(* IEC 61131-3 sources: volt/packages/volt-lsp-iec/test-corpus/pro2193/Device/Plc Logic/Application/05 Global Var Lists, 12 files *)

(* ---- enumExchangeSets.dut ---- *)
{attribute 'qualified_only'}
{attribute 'strict'}
{attribute 'to_string'}
TYPE enumExchangeSets :
(
	Default
//	SingleCavSingleTakeover,
//	SingleCavDualTakeover,
//	FourCavDualTakeover,
//	TwoCavSingleTakeover
);
END_TYPE

// Please rename 'Default' to a more descriptive name.
// Check the type plate on the gripper how it is named.

// HINT!! Right-click on 'Default' -> Refactoring -> Rename ...

(* ---- RetainedVarsInBrinkRecipeType.dut ---- *)
// Retained variables that are saved in the Brink recipe. These are not changed when the customer picks a new recipe.
{attribute 'symbol' := 'readwrite'}
TYPE RetainedVarsInBrinkRecipeType :
STRUCT
	maximumAllowedCycleTime	: IntWithLimitsType	:=		// Time (sec) after which 'maximum allowed cycle time exceeded' alarm trips.
	(
		lowerLimit	:= 10,
		value		:= 30,
		upperLimit	:= 300,
		stepSize	:= 10
	);

	machineIdleShutoffTime	: IntWithLimitsType :=		// Time (min) when machine is inactive, shut off main air valve and vacuumpumps.
	(
		lowerLimit	:= 5,
		value		:= 30,
		upperLimit	:= 60 * 24 * 7,
		stepSize	:= 10
	);

	workingLightsTime		: IntWithLimitsType :=		// Time (min) that working lights will illuminate the inside of the machine.
	(
		lowerLimit	:= 5,
		value		:= 30,
		upperLimit	:= 60 * 24 * 7,
		stepSize	:= 5
	);

	// When the Xi Unit needs a label, and the magazine has no label ready: Wait for the label to be ready? Or check again the next cycle.
	// The process will wait for new labels for this time. After time-out the cycle continues without a label.
	cycleContinuesWithoutLabelsAfterTimeout		: RealWithLimitsType :=
	(
		lowerLimit	:= 0,						// Set to 0 to never wait for the magazine
		value		:= 10,
		upperLimit	:= 60.0 * 60.0 * 24,		// Set to 60*60*24 to wait the whole day
		stepSize	:= 1
	);

END_STRUCT
END_TYPE

(* ---- RetainedVarsInRecipeType.dut ---- *)
// Retained variables that are saved in the customer recipe
{attribute 'symbol' := 'readwrite'}
TYPE RetainedVarsInRecipeType :
STRUCT
	// Read only variables for safety. Vars can be changed by buttons in HMI program.
	{attribute 'symbol' := 'read'}	EnableIML					: BOOL;
	{attribute 'symbol' := 'read'}	EnableHMU					: BOOL;
	{attribute 'symbol' := 'read'}	EnableVision				: BOOL;
	{attribute 'symbol' := 'read'}	EnableSticker				: BOOL;

	ActiveExchangeSet			: enumExchangeSets;

	targetCycleTime				: REAL;	// The desired cycle time (sec) for this recipe. Used for statistics.

	productWeight				: REAL;	// Weight of a single product as measured by the customer (g).

	productPitch				: RealWithLimitsType :=		// Pitch between the products (mm).
	(
		lowerLimit	:= 0.1,
		value		:= 0.1,
		upperLimit	:= 100,
		stepSize	:= 0.1
	);

	productHeight				: RealWithLimitsType :=		// Height of a single product (mm).
	(
		lowerLimit	:= 1,
		value		:= 1,
		upperLimit	:= 500,
		stepSize	:= 2
	);

	{attribute 'symbol' := 'none'}	chainPos_XuUnit				: ARRAY[1..GVL_Constants.ChainProductsForXuUnit] OF UINT;
	{attribute 'symbol' := 'none'}	chainPos_Camera				: UINT;
	{attribute 'symbol' := 'none'}	chainPos_Reject				: ARRAY[1..GVL_Constants.ChainProductsForReject] OF UINT;
	{attribute 'symbol' := 'none'}	chainPos_ZUnit				: ARRAY[1..GVL_Constants.ChainProductsForZUnit] OF UINT;
	{attribute 'symbol' := 'none'}	chainPos_Sensor				: UINT;

END_STRUCT
END_TYPE

(* ---- GlobalVars.gvl ---- *)
{attribute 'symbol' := 'none'}
{attribute 'qualified_only'}
{attribute 'analysis' := '-33'}	// Unused Variable
VAR_GLOBAL
	Reset					: BOOL;					// Global reset active. From hardware button or input from visualisation
	EnableServoDrives		: BOOL;
	EnableMainvalve			: BOOL;
	manualControlRequested	: BOOL;					// Is high when a manual control button was pushed on the HMI

	BlinkerNormal			: BOOL;					// Global blinking bool. Default: high for 0,5 sec.
	BlinkerFast				: BOOL;					// Global fast blinker. Default: high for 0.2 sec.
	BlinkerPulseFast		: BOOL;					// Used by gates. Fast 0.1 sec. pulses
	BlinkerPulseSlow		: BOOL;					// Used by gates. Slow 0.1 sec. pulses

	EmergencyStopActive		: BOOL;					// Emergency-stop is active.

	debugTestBool1			: BOOL;
	debugTestBool2			: BOOL;
	debugTestInt1			: INT;
	debugTestInt2			: INT;
	debugTestInt3			: INT;
	debugTestInt4			: INT;
	debugTestInt5			: INT;
	debugSW					: ARRAY[0..9] OF StopwatchFB;

	// SUBRANGE not supported by VisiWinNet :(
	{attribute 'symbol' := 'readwrite'}	ActMouldLevels			: UINT(*(1..GVL_Constants.MaxMouldLevels)*)	:= GVL_Constants.MaxMouldLevels;
	{attribute 'symbol' := 'readwrite'}	ActProductsInX			: UINT(*(1..GVL_Constants.MaxProductsInX)*)	:= GVL_Constants.MaxProductsInX;
	{attribute 'symbol' := 'readwrite'}	ActProductsInY			: UINT(*(1..GVL_Constants.MaxProductsInY)*)	:= GVL_Constants.MaxProductsInY;
	ActProductsInMould		: UINT	:= ActMouldLevels * ActProductsInX * ActProductsInY;

	fbModuleManager			: ModuleManagerFB(name := 'SER');	// Keep a record of different kinds of modules in the machine.

	immediatelyGetNewLabels	: BOOL;					// In semi-auto mode, new labels are taken from magazine only AFTER the labels are inserted in the mould. This can overide that behaviouw.

	RuntimeConstants		: RuntimeConstantsType;	// For debugging: some constants about the PLC.

	// Options for debugging
	CheckBoundFunctionsThrowExceptions	: BOOL := FALSE;	// When the CheckBounds function has an error, the PLC is stopped. This makes troubleshooting easier.
	EnableDebugLogging					: BOOL := FALSE;	// Debug log messages are disabled and NOT logged to the PLC.
	EnableLoggingAllStateChanges		: BOOL := FALSE;	// Create a log message for every state change
	activeAlarmInstance					: STRING(80);		// For debugging: show id of module that has an alarm active
END_VAR

(* ---- GlobalVars_BFU.gvl ---- *)
{attribute 'symbol' := 'none'}
{attribute 'qualified_only'}
{attribute 'analysis' := '-33'}	// Unused Variable
VAR_GLOBAL
	Reset					: BOOL;					// Global reset active. From hardware button or input from visualisation
	EnableMainvalve			: BOOL;
	EnableServoDrives		: BOOL;

	fbModuleManager			: ModuleManagerFB(name := 'BFU');	// Keep a record of different kinds of modules in the machine.
END_VAR

(* ---- GVL_ComponentHardware.gvl ---- *)
(* This code is generated automatically *)
(* Don't change the content! *)

{attribute 'qualified_only'}
{attribute 'linkalways'}
VAR_GLOBAL
	//Controller
	Device 	: L_IC1P_ComponentHardware;

	//EtherCAT device
	L_i750_ZR 	: L_IC1P_ComponentHardware;
	L_i750_C2 	: L_IC1P_ComponentHardware;
	L_i750_M1 	: L_IC1P_ComponentHardware;
	L_i750_M2 	: L_IC1P_ComponentHardware;
	L_i750_Z 	: L_IC1P_ComponentHardware;
	L_i750_C1 	: L_IC1P_ComponentHardware;
	L_i750_Xi 	: L_IC1P_ComponentHardware;
	L_i750_Xu 	: L_IC1P_ComponentHardware;
	L_i950_Y 	: L_IC1P_ComponentHardware;
	RIO_M1 	: L_IC1P_ComponentHardware;
	RIO_Z1 	: L_IC1P_ComponentHardware;
	RIO_BFU 	: L_IC1P_ComponentHardware;
	FANUC_R_30iB_Plus 	: L_IC1P_ComponentHardware;

	//I/O module
	DI_30 	: L_IC1P_ComponentHardware;
	DI_31 	: L_IC1P_ComponentHardware;
	DI_32 	: L_IC1P_ComponentHardware;
	DI_33 	: L_IC1P_ComponentHardware;
	DQ_30 	: L_IC1P_ComponentHardware;
	DQ_31 	: L_IC1P_ComponentHardware;
	DQ_32 	: L_IC1P_ComponentHardware;
	DQ_33 	: L_IC1P_ComponentHardware;
	DQ_34 	: L_IC1P_ComponentHardware;
	DQ_35 	: L_IC1P_ComponentHardware;
	DQ_36 	: L_IC1P_ComponentHardware;
	DI_40 	: L_IC1P_ComponentHardware;
	DI_41 	: L_IC1P_ComponentHardware;
	DI_42 	: L_IC1P_ComponentHardware;
	DI_43 	: L_IC1P_ComponentHardware;
	DI_44 	: L_IC1P_ComponentHardware;
	DI_45 	: L_IC1P_ComponentHardware;
	DQ_40 	: L_IC1P_ComponentHardware;
	DQ_41 	: L_IC1P_ComponentHardware;
	DQ_42 	: L_IC1P_ComponentHardware;
	DQ_43 	: L_IC1P_ComponentHardware;
	DQ_44 	: L_IC1P_ComponentHardware;
	DQ_45 	: L_IC1P_ComponentHardware;
	DQ_46 	: L_IC1P_ComponentHardware;
	DI_50 	: L_IC1P_ComponentHardware;
	DI_51 	: L_IC1P_ComponentHardware;
	DI_52 	: L_IC1P_ComponentHardware;
	DI_53 	: L_IC1P_ComponentHardware;
	DI_54 	: L_IC1P_ComponentHardware;
	DQ_50 	: L_IC1P_ComponentHardware;
	DQ_51 	: L_IC1P_ComponentHardware;
	DQ_52 	: L_IC1P_ComponentHardware;
	DQ_53 	: L_IC1P_ComponentHardware;
	DQ_54 	: L_IC1P_ComponentHardware;

END_VAR

(* ---- GVL_Constants.gvl ---- *)
{attribute 'qualified_only'}
{attribute 'analysis' := '-33'}	// Unused Variable
VAR_GLOBAL CONSTANT
	MaxRejectReasonsMisc		: USINT			:= 1;		// IMM Euromap Reject, handle mounting reject, mould measurement reject, etc.
	MaxRejectReasonsCamera		: USINT			:= 7;		// Cam1 Reject, Cam2 Reject, etc.
	MaxRejectReasonsTotal		: USINT			:= MaxRejectReasonsMisc + MaxRejectReasonsCamera;

	MaxMouldLevels				: UINT			:= 1;		// In case of a stack mould, the number of mould faces (or levels)
	MaxProductsInX				: UINT			:= 3;		// Number of cavities in mould in X direction (horizontal)
	MaxProductsInY				: UINT			:= 4;		// Number of cavities in mould in Y direction (vertical)
	MaxProductsInMould			: UINT			:= MaxMouldLevels * MaxProductsInX * MaxProductsInY;	// Total number of cavities

	CavityStartIndex			: UINT			:= 1;											// Cavity numbering start index (usually 1)
	CavityEndIndex				: UINT			:= CavityStartIndex - 1 + MaxProductsInMould;	// Cavity numbering end index (usually the same as MaxProductsInMould)

	ChainProductsForXuUnit		: USINT			:= 4;
	ChainProductsForReject		: USINT			:= 1;
	ChainProductsForZUnit		: USINT			:= 6;
	ZUnitProductsForConveyor	: USINT			:= 12;

	ArmLength					: REAL			:= 895.0;	// Length of the arm/gripper in the drawer magazine in mm, normally 895 mm
	MaxAttemptsLabelTakeOut		: UINT			:= 1;		// Number of times the magazine attempts to take a label before assuming that the magazine is empty

	// Constants for Recipe Management
	RecipeDefinitionsCount		: INT			:= 3;		// Number of different recipe definitions
	AllRecipeDefinitions		: ARRAY[1..RecipeDefinitionsCount] OF STRING := ['Brink', 'Customer', 'Cassette'];	// Names of recipe definitions that are added to the Recipe Manager

	// Constants for Module Manager
	MaxNumberOfModules			: UINT			:= 40;		// Maximum amount of modules that the machine may have.
	MaxNumberOfStartableModules	: UINT			:= 20;		// Maximum amount of startable modules
	MaxNumberOfResettableModules: UINT			:= 20;		// Maximum amount of resettable modules
	MaxNumberOfServoDrives		: UINT			:= 20;		// Maximum amount of servo drives
	MaxNumberOfGates			: UINT			:= 10;		// Maximum amount of safety gates

	TimeLongest					: TIME			:= T#49D17H2M47S295MS;				// 4294967295
	DateTimeEarliest			: DATE_AND_TIME	:= DATE_AND_TIME#1970-1-1-00:00:00;	// 0
	DateTimeLatest				: DATE_AND_TIME	:= DATE_AND_TIME#2106-2-7-6:28:15;	// 4294967295

	RealSmallest				: REAL			:= -3.402823E+38;					// Smallest number
	RealLargest					: REAL			:=  3.402823E+38;					// Largest number
	LRealSmallest				: LREAL			:= -1.7976931348623157E+308;		// Smallest number
	LRealLargest				: LREAL			:=  1.7976931348623157E+308;		// Largest number
	DintSmallest				: DINT			:= -2147483648;						// Lower limit of DINT datatype
	DintLargest					: DINT			:=  2147483647;						// Upper limit of DINT datatype
	pi							: REAL			:= 3.14159274101257324;				// π
END_VAR

(* ---- GVL_Constants_BFU.gvl ---- *)
{attribute 'qualified_only'}
{attribute 'analysis' := '-33'}	// Unused Variable
VAR_GLOBAL CONSTANT
	MaxNumberOfStacksInBox		: UINT	:= 30;		// Maximum allowed number of stacks in the box

	// Constants for Module Manager
	MaxNumberOfModules			: UINT	:= 40;		// Maximum amount of modules that the machine may have.
	MaxNumberOfStartableModules	: UINT	:= 20;		// Maximum amount of startable modules
	MaxNumberOfResettableModules: UINT	:= 20;		// Maximum amount of resettable modules
	MaxNumberOfServoDrives		: UINT	:= 20;		// Maximum amount of servo drives
	MaxNumberOfGates			: UINT	:= 10;		// Maximum amount of safety gates
END_VAR

(* ---- GVL_Constants_Magazine.gvl ---- *)
{attribute 'qualified_only'}
VAR_GLOBAL CONSTANT
	MaxCassettes		: USINT := 16;
	MaxEnableValves		: USINT	:= 8;
	MaxAdjustValves		: USINT := 6;

	// Table defining all motors and directions for all possible combinations of label and cassette orientations
	OrientationTable	: ARRAY[1..64] OF OrientationEntry :=
	[
		(CassetteOrientation := enumOrientationType.Upright,	LabelOrientation := enumOrientationType.Upright,	Movement := enumMovementType.Up,	Motor := enumMotorsType.X,	Direction := enumdirection.Positive),
		(CassetteOrientation := enumOrientationType.Upright,	LabelOrientation := enumOrientationType.Upright,	Movement := enumMovementType.Down,	Motor := enumMotorsType.X,	Direction := enumDirection.Negative),
		(CassetteOrientation := enumOrientationType.Upright,	LabelOrientation := enumOrientationType.Upright,	Movement := enumMovementType.Left,	Motor := enumMotorsType.Y,	Direction := enumDirection.Negative),
		(CassetteOrientation := enumOrientationType.Upright,	LabelOrientation := enumOrientationType.Upright,	Movement := enumMovementType.Right,	Motor := enumMotorsType.Y,	Direction := enumDirection.Positive),
		(CassetteOrientation := enumOrientationType.Upright,	LabelOrientation := enumOrientationType.Right,		Movement := enumMovementType.Up,	Motor := enumMotorsType.Y,	Direction := enumDirection.Positive),
		(CassetteOrientation := enumOrientationType.Upright,	LabelOrientation := enumOrientationType.Right,		Movement := enumMovementType.Down,	Motor := enumMotorsType.Y,	Direction := enumDirection.Negative),
		(CassetteOrientation := enumOrientationType.Upright,	LabelOrientation := enumOrientationType.Right,		Movement := enumMovementType.Left,	Motor := enumMotorsType.X,	Direction := enumDirection.Positive),
		(CassetteOrientation := enumOrientationType.Upright,	LabelOrientation := enumOrientationType.Right,		Movement := enumMovementType.Right,	Motor := enumMotorsType.X,	Direction := enumDirection.Negative),
		(CassetteOrientation := enumOrientationType.Upright,	LabelOrientation := enumOrientationType.UpsideDown,	Movement := enumMovementType.Up,	Motor := enumMotorsType.X,	Direction := enumDirection.Negative),
		(CassetteOrientation := enumOrientationType.Upright,	LabelOrientation := enumOrientationType.UpsideDown,	Movement := enumMovementType.Down,	Motor := enumMotorsType.X,	Direction := enumDirection.Positive),
		(CassetteOrientation := enumOrientationType.Upright,	LabelOrientation := enumOrientationType.UpsideDown,	Movement := enumMovementType.Left,	Motor := enumMotorsType.Y,	Direction := enumDirection.Positive),
		(CassetteOrientation := enumOrientationType.Upright,	LabelOrientation := enumOrientationType.UpsideDown,	Movement := enumMovementType.Right,	Motor := enumMotorsType.Y,	Direction := enumDirection.Negative),
		(CassetteOrientation := enumOrientationType.Upright,	LabelOrientation := enumOrientationType.Left,		Movement := enumMovementType.Up,	Motor := enumMotorsType.Y,	Direction := enumDirection.Negative),
		(CassetteOrientation := enumOrientationType.Upright,	LabelOrientation := enumOrientationType.Left,		Movement := enumMovementType.Down,	Motor := enumMotorsType.Y,	Direction := enumDirection.Positive),
		(CassetteOrientation := enumOrientationType.Upright,	LabelOrientation := enumOrientationType.Left,		Movement := enumMovementType.Left,	Motor := enumMotorsType.X,	Direction := enumDirection.Negative),
		(CassetteOrientation := enumOrientationType.Upright,	LabelOrientation := enumOrientationType.Left,		Movement := enumMovementType.Right,	Motor := enumMotorsType.X,	Direction := enumDirection.Positive),
		(CassetteOrientation := enumOrientationType.Right,		LabelOrientation := enumOrientationType.Upright,	Movement := enumMovementType.Up,	Motor := enumMotorsType.Y,	Direction := enumDirection.Negative),
		(CassetteOrientation := enumOrientationType.Right,		LabelOrientation := enumOrientationType.Upright,	Movement := enumMovementType.Down,	Motor := enumMotorsType.Y,	Direction := enumDirection.Positive),
		(CassetteOrientation := enumOrientationType.Right,		LabelOrientation := enumOrientationType.Upright,	Movement := enumMovementType.Left,	Motor := enumMotorsType.X,	Direction := enumDirection.Negative),
		(CassetteOrientation := enumOrientationType.Right,		LabelOrientation := enumOrientationType.Upright,	Movement := enumMovementType.Right,	Motor := enumMotorsType.X,	Direction := enumDirection.Positive),
		(CassetteOrientation := enumOrientationType.Right,		LabelOrientation := enumOrientationType.Right,		Movement := enumMovementType.Up,	Motor := enumMotorsType.X,	Direction := enumDirection.Positive),
		(CassetteOrientation := enumOrientationType.Right,		LabelOrientation := enumOrientationType.Right,		Movement := enumMovementType.Down,	Motor := enumMotorsType.X,	Direction := enumDirection.Negative),
		(CassetteOrientation := enumOrientationType.Right,		LabelOrientation := enumOrientationType.Right,		Movement := enumMovementType.Left,	Motor := enumMotorsType.Y,	Direction := enumDirection.Negative),
		(CassetteOrientation := enumOrientationType.Right,		LabelOrientation := enumOrientationType.Right,		Movement := enumMovementType.Right,	Motor := enumMotorsType.Y,	Direction := enumDirection.Positive),
		(CassetteOrientation := enumOrientationType.Right,		LabelOrientation := enumOrientationType.UpsideDown,	Movement := enumMovementType.Up,	Motor := enumMotorsType.Y,	Direction := enumDirection.Positive),
		(CassetteOrientation := enumOrientationType.Right,		LabelOrientation := enumOrientationType.UpsideDown,	Movement := enumMovementType.Down,	Motor := enumMotorsType.Y,	Direction := enumDirection.Negative),
		(CassetteOrientation := enumOrientationType.Right,		LabelOrientation := enumOrientationType.UpsideDown,	Movement := enumMovementType.Left,	Motor := enumMotorsType.X,	Direction := enumDirection.Positive),
		(CassetteOrientation := enumOrientationType.Right,		LabelOrientation := enumOrientationType.UpsideDown,	Movement := enumMovementType.Right,	Motor := enumMotorsType.X,	Direction := enumDirection.Negative),
		(CassetteOrientation := enumOrientationType.Right,		LabelOrientation := enumOrientationType.Left,		Movement := enumMovementType.Up,	Motor := enumMotorsType.X,	Direction := enumDirection.Negative),
		(CassetteOrientation := enumOrientationType.Right,		LabelOrientation := enumOrientationType.Left,		Movement := enumMovementType.Down,	Motor := enumMotorsType.X,	Direction := enumDirection.Positive),
		(CassetteOrientation := enumOrientationType.Right,		LabelOrientation := enumOrientationType.Left,		Movement := enumMovementType.Left,	Motor := enumMotorsType.Y,	Direction := enumDirection.Positive),
		(CassetteOrientation := enumOrientationType.Right,		LabelOrientation := enumOrientationType.Left,		Movement := enumMovementType.Right,	Motor := enumMotorsType.Y,	Direction := enumDirection.Negative),
		(CassetteOrientation := enumOrientationType.UpsideDown,	LabelOrientation := enumOrientationType.Upright,	Movement := enumMovementType.Up,	Motor := enumMotorsType.X,	Direction := enumDirection.Negative),
		(CassetteOrientation := enumOrientationType.UpsideDown,	LabelOrientation := enumOrientationType.Upright,	Movement := enumMovementType.Down,	Motor := enumMotorsType.X,	Direction := enumDirection.Positive),
		(CassetteOrientation := enumOrientationType.UpsideDown,	LabelOrientation := enumOrientationType.Upright,	Movement := enumMovementType.Left,	Motor := enumMotorsType.Y,	Direction := enumDirection.Positive),
		(CassetteOrientation := enumOrientationType.UpsideDown,	LabelOrientation := enumOrientationType.Upright,	Movement := enumMovementType.Right,	Motor := enumMotorsType.Y,	Direction := enumDirection.Negative),
		(CassetteOrientation := enumOrientationType.UpsideDown,	LabelOrientation := enumOrientationType.Right,		Movement := enumMovementType.Up,	Motor := enumMotorsType.Y,	Direction := enumDirection.Negative),
		(CassetteOrientation := enumOrientationType.UpsideDown,	LabelOrientation := enumOrientationType.Right,		Movement := enumMovementType.Down,	Motor := enumMotorsType.Y,	Direction := enumDirection.Positive),
		(CassetteOrientation := enumOrientationType.UpsideDown,	LabelOrientation := enumOrientationType.Right,		Movement := enumMovementType.Left,	Motor := enumMotorsType.X,	Direction := enumDirection.Negative),
		(CassetteOrientation := enumOrientationType.UpsideDown,	LabelOrientation := enumOrientationType.Right,		Movement := enumMovementType.Right,	Motor := enumMotorsType.X,	Direction := enumDirection.Positive),
		(CassetteOrientation := enumOrientationType.UpsideDown,	LabelOrientation := enumOrientationType.UpsideDown,	Movement := enumMovementType.Up,	Motor := enumMotorsType.X,	Direction := enumDirection.Positive),
		(CassetteOrientation := enumOrientationType.UpsideDown,	LabelOrientation := enumOrientationType.UpsideDown,	Movement := enumMovementType.Down,	Motor := enumMotorsType.X,	Direction := enumDirection.Negative),
		(CassetteOrientation := enumOrientationType.UpsideDown,	LabelOrientation := enumOrientationType.UpsideDown,	Movement := enumMovementType.Left,	Motor := enumMotorsType.Y,	Direction := enumDirection.Negative),
		(CassetteOrientation := enumOrientationType.UpsideDown,	LabelOrientation := enumOrientationType.UpsideDown,	Movement := enumMovementType.Right,	Motor := enumMotorsType.Y,	Direction := enumDirection.Positive),
		(CassetteOrientation := enumOrientationType.UpsideDown,	LabelOrientation := enumOrientationType.Left,		Movement := enumMovementType.Up,	Motor := enumMotorsType.Y,	Direction := enumDirection.Positive),
		(CassetteOrientation := enumOrientationType.UpsideDown,	LabelOrientation := enumOrientationType.Left,		Movement := enumMovementType.Down,	Motor := enumMotorsType.Y,	Direction := enumDirection.Negative),
		(CassetteOrientation := enumOrientationType.UpsideDown,	LabelOrientation := enumOrientationType.Left,		Movement := enumMovementType.Left,	Motor := enumMotorsType.X,	Direction := enumDirection.Positive),
		(CassetteOrientation := enumOrientationType.UpsideDown,	LabelOrientation := enumOrientationType.Left,		Movement := enumMovementType.Right,	Motor := enumMotorsType.X,	Direction := enumDirection.Negative),
		(CassetteOrientation := enumOrientationType.Left,		LabelOrientation := enumOrientationType.Upright,	Movement := enumMovementType.Up,	Motor := enumMotorsType.Y,	Direction := enumDirection.Positive),
		(CassetteOrientation := enumOrientationType.Left,		LabelOrientation := enumOrientationType.Upright,	Movement := enumMovementType.Down,	Motor := enumMotorsType.Y,	Direction := enumDirection.Negative),
		(CassetteOrientation := enumOrientationType.Left,		LabelOrientation := enumOrientationType.Upright,	Movement := enumMovementType.Left,	Motor := enumMotorsType.X,	Direction := enumDirection.Positive),
		(CassetteOrientation := enumOrientationType.Left,		LabelOrientation := enumOrientationType.Upright,	Movement := enumMovementType.Right,	Motor := enumMotorsType.X,	Direction := enumDirection.Negative),
		(CassetteOrientation := enumOrientationType.Left,		LabelOrientation := enumOrientationType.Right,		Movement := enumMovementType.Up,	Motor := enumMotorsType.X,	Direction := enumDirection.Negative),
		(CassetteOrientation := enumOrientationType.Left,		LabelOrientation := enumOrientationType.Right,		Movement := enumMovementType.Down,	Motor := enumMotorsType.X,	Direction := enumDirection.Positive),
		(CassetteOrientation := enumOrientationType.Left,		LabelOrientation := enumOrientationType.Right,		Movement := enumMovementType.Left,	Motor := enumMotorsType.Y,	Direction := enumDirection.Positive),
		(CassetteOrientation := enumOrientationType.Left,		LabelOrientation := enumOrientationType.Right,		Movement := enumMovementType.Right,	Motor := enumMotorsType.Y,	Direction := enumDirection.Negative),
		(CassetteOrientation := enumOrientationType.Left,		LabelOrientation := enumOrientationType.UpsideDown,	Movement := enumMovementType.Up,	Motor := enumMotorsType.Y,	Direction := enumDirection.Negative),
		(CassetteOrientation := enumOrientationType.Left,		LabelOrientation := enumOrientationType.UpsideDown,	Movement := enumMovementType.Down,	Motor := enumMotorsType.Y,	Direction := enumDirection.Positive),
		(CassetteOrientation := enumOrientationType.Left,		LabelOrientation := enumOrientationType.UpsideDown,	Movement := enumMovementType.Left,	Motor := enumMotorsType.X,	Direction := enumDirection.Negative),
		(CassetteOrientation := enumOrientationType.Left,		LabelOrientation := enumOrientationType.UpsideDown,	Movement := enumMovementType.Right,	Motor := enumMotorsType.X,	Direction := enumDirection.Positive),
		(CassetteOrientation := enumOrientationType.Left,		LabelOrientation := enumOrientationType.Left,		Movement := enumMovementType.Up,	Motor := enumMotorsType.X,	Direction := enumDirection.Positive),
		(CassetteOrientation := enumOrientationType.Left,		LabelOrientation := enumOrientationType.Left,		Movement := enumMovementType.Down,	Motor := enumMotorsType.X,	Direction := enumDirection.Negative),
		(CassetteOrientation := enumOrientationType.Left,		LabelOrientation := enumOrientationType.Left,		Movement := enumMovementType.Left,	Motor := enumMotorsType.Y,	Direction := enumDirection.Negative),
		(CassetteOrientation := enumOrientationType.Left,		LabelOrientation := enumOrientationType.Left,		Movement := enumMovementType.Right,	Motor := enumMotorsType.Y,	Direction := enumDirection.Positive)
	];
END_VAR

(* ---- GVL_HC.gvl ---- *)
(* This code is generated automatically *)
(* Don't change the content! *)

{attribute 'qualified_only'}
{attribute 'linkalways'}
VAR_GLOBAL
	HcGroups : ARRAY [0..1] OF L_ETC_HC_GROUP;
END_VAR

(* ---- GVL_VacuumNumbers.gvl ---- *)
{attribute 'analysis' := '-33'}	// Unused Variable
VAR_GLOBAL CONSTANT
	// Use the constants below to access bits in any integer parameter
	AllVacuums			: WORD := 0;	// Ask all vacuums (parameter is zero)
	Vacuum00			: WORD := 0;	// Vacuum 0 (first bit) will not be in use! Vacuums start numbering from 1.
	Vacuum01			: WORD := 1;	// Ask vacuum 1 (or products belonging to vacuum 1)
	Vacuum02			: WORD := 2;	// Ask vacuum 2 (or products belonging to vacuum 2)
	Vacuum03			: WORD := 3;	// Ask vacuum 3 (or products belonging to vacuum 3)
	Vacuum04			: WORD := 4;	// Ask vacuum 4 (or products belonging to vacuum 4)
	Vacuum05			: WORD := 5;	// Ask vacuum 5 (or products belonging to vacuum 5)
	Vacuum06			: WORD := 6;	// Ask vacuum 6 (or products belonging to vacuum 6)
	Vacuum07			: WORD := 7;	// Ask vacuum 7 (or products belonging to vacuum 7)
	Vacuum08			: WORD := 8;	// Ask vacuum 8 (or products belonging to vacuum 8)
	Vacuum09			: WORD := 9;	// Ask vacuum 9 (or products belonging to vacuum 9)
	Vacuum10			: WORD := 10;	// Ask vacuum 10 (or products belonging to vacuum 10)
	Vacuum11			: WORD := 11;	// Ask vacuum 11 (or products belonging to vacuum 11)
	Vacuum12			: WORD := 12;	// Ask vacuum 12 (or products belonging to vacuum 12)
	Vacuum13			: WORD := 13;	// Ask vacuum 13 (or products belonging to vacuum 13)
	Vacuum14			: WORD := 14;	// Ask vacuum 14 (or products belonging to vacuum 14)
	Vacuum15			: WORD := 15;	// Ask vacuum 15 (or products belonging to vacuum 15)
END_VAR

// So to access the second bit in an integer, use like this:
// vacuumIndex.Vacuum01 := true;

// No 'qualified_only' attribute! Or bitaccess doesn't work.

(* ---- PersistentVars.gvl ---- *)
{attribute 'qualified_only'}
{attribute 'symbol' := 'readwrite'}
VAR_GLOBAL PERSISTENT RETAIN
	RecipeVars						: RetainedVarsInRecipeType;
	BrinkRecipeVars					: RetainedVarsInBrinkRecipeType;

	disableBuzzer					: BOOL;					// Permanently disable the buzzer output

	// SUBRANGE not supported by VisiWinNet :(
	usiGlobalSERSpeed				: USINT(*(1..100)*) := 50;	// Limit speed of all drives in the SER robot (0 to 100%)
	usiGlobalBFUSpeed				: USINT(*(1..100)*) := 50;	// Limit speed of all drives in the BFU robot (0 to 100%)

	DisableVacuumWithAirButton		: BOOL := FALSE;
	DisableVacuumPump2				: BOOL;

	{attribute 'symbol' := 'none'}	vacuumPumpRunningTime		: UDINT;				// Total time the vacuumpump has been running.
	{attribute 'symbol' := 'none'}	vacuumPumpNumberOfStarts	: UDINT;				// Total number of times the vacuumpump has been started.
	{attribute 'symbol' := 'none'}	Statistics					: ARRAY[1..ProductionStatsFB.NumberOfStatisticSets] OF ProductionStatsType;

	rejectReasonDescriptions		: ARRAY[1..GVL_Constants.MaxRejectReasonsTotal] OF STRING(40) :=
	[
		'IMM Euromap Reject',		// 1
		'Cam 1 Reject',				// 2
		'Cam 2 Reject',				// 3
		'Cam 3 Reject',				// 4
		'Cam 4 Reject',				// 5
		'Cam 5 Reject',				// 6
		'Cam 6 Reject',				// 7
		'Cam 7 Reject'				// 8
	];

	{attribute 'symbol' := 'none'}	cavityAliases				: ARRAY[GVL_Constants.CavityStartIndex..GVL_Constants.CavityEndIndex] OF STRING(20);

	// Generated instance path of persistent variable
	CassetteAdjustments.Data: ARRAY [1..CassetteAdjustments.usiNumberOfUnits] OF ARRAY [enumDrawer.Upper..enumDrawer.Lower, 1..GVL_Constants_Magazine.MaxCassettes] OF CassettePosition;
	// Generated instance path of persistent variable
	CassetteAdjustments.SwitchCountEnable: ARRAY [1..CassetteAdjustments.usiNumberOfUnits] OF ARRAY [enumDrawer.Upper..enumDrawer.Lower, 1..GVL_Constants_Magazine.MaxEnableValves] OF UDINT;
	// Generated instance path of persistent variable
	CassetteAdjustments.SwitchCountAdjust: ARRAY [1..CassetteAdjustments.usiNumberOfUnits] OF ARRAY [enumDrawer.Upper..enumDrawer.Lower, 1..GVL_Constants_Magazine.MaxAdjustValves] OF UDINT;
	// Generated instance path of persistent variable
	CassetteAdjustments.SwitchCountCassette: ARRAY [1..CassetteAdjustments.usiNumberOfUnits] OF ARRAY [enumDrawer.Upper..enumDrawer.Lower, 1..GVL_Constants_Magazine.MaxCassettes] OF ARRAY [enumMotorsType.X1..enumMotorsType.Y] OF UDINT;
	// Generated instance path of persistent variable
	CassetteAdjustments.ActualCassettePosition: ARRAY [1..CassetteAdjustments.usiNumberOfUnits] OF ARRAY [enumDrawer.Upper..enumDrawer.Lower, 1..GVL_Constants_Magazine.MaxCassettes] OF CassettePosition;
	// Generated instance path of persistent variable
	CassetteAdjustments.TargetCassettePosition: ARRAY [1..CassetteAdjustments.usiNumberOfUnits] OF ARRAY [enumDrawer.Upper..enumDrawer.Lower, 1..GVL_Constants_Magazine.MaxCassettes] OF CassettePosition;
	// Generated instance path of persistent variable
	RecipeControl.activeRecipe: ARRAY [1..GVL_Constants.RecipeDefinitionsCount] OF STRING(80);
	// Generated instance path of persistent variable
	RecipeControl.MetaData: ARRAY [1..GVL_Constants.RecipeDefinitionsCount] OF RecipeMetaDataType;
	// Generated instance path of persistent variable
	Fanucs.Data: ARRAY [1..Fanucs.usiNumberOfUnits] OF FanucUnitBase_Data;
	// Generated instance path of persistent variable
	Fanucs.DataProject: ARRAY [1..Fanucs.usiNumberOfUnits] OF FanucUnit_Data;
	// Generated instance path of persistent variable
	Fanucs.GripperStatus: ARRAY [1..Fanucs.usiNumberOfUnits] OF StackStatusType;
	// Generated instance path of persistent variable
	YUnits.Data: ARRAY [1..YUnits.usiNumberOfUnits] OF YUnit_Default_Data;
	// Generated instance path of persistent variable
	YUnits.DataBrink: ARRAY [1..YUnits.usiNumberOfUnits] OF DataBrinkType;
	// Generated instance path of persistent variable
	YUnits.coveredDistance: ARRAY [1..YUnits.usiNumberOfUnits] OF UDINT;
	// Generated instance path of persistent variable
	XuUnits.Data: ARRAY [1..XuUnits.usiNumberOfUnits] OF XuUnit_Default_Data;
	// Generated instance path of persistent variable
	XuUnits.DataProject: ARRAY [1..XuUnits.usiNumberOfUnits] OF XuUnit_ForChain_Data;
	// Generated instance path of persistent variable
	XuUnits.DataBrink: ARRAY [1..XuUnits.usiNumberOfUnits] OF DataBrinkType;
	// Generated instance path of persistent variable
	XuUnits.coveredDistance: ARRAY [1..XuUnits.usiNumberOfUnits] OF UDINT;
	// Generated instance path of persistent variable
	ZUnits.Data: ARRAY [1..ZUnits.usiNumberOfUnits] OF ZUnit_Base_Data;
	// Generated instance path of persistent variable
	ZUnits.DataProject: ARRAY [1..ZUnits.usiNumberOfUnits] OF ZUnit_ForChainWithServoRotate_Data;
	// Generated instance path of persistent variable
	ZUnits.DataBrink: ARRAY [1..ZUnits.usiNumberOfUnits] OF DataBrinkType;
	// Generated instance path of persistent variable
	ZUnits.coveredDistance: ARRAY [1..ZUnits.usiNumberOfUnits] OF UDINT;
	// Generated instance path of persistent variable
	XiUnits.Data: ARRAY [1..XiUnits.usiNumberOfUnits] OF XiUnit_Default_Data;
	// Generated instance path of persistent variable
	XiUnits.DataProject: ARRAY [1..XiUnits.usiNumberOfUnits] OF XiUnit_Data;
	// Generated instance path of persistent variable
	XiUnits.DataBrink: ARRAY [1..XiUnits.usiNumberOfUnits] OF DataBrinkType;
	// Generated instance path of persistent variable
	XiUnits.coveredDistance: ARRAY [1..XiUnits.usiNumberOfUnits] OF UDINT;
	// Generated instance path of persistent variable
	ZRUnits.Data: ARRAY [1..ZRUnits.usiNumberOfUnits] OF ZRUnit_Default_Data;
	// Generated instance path of persistent variable
	ZRUnits.DataBrink: ARRAY [1..ZRUnits.usiNumberOfUnits] OF DataBrinkType;
	// Generated instance path of persistent variable
	ZRUnits.coveredDistance: ARRAY [1..ZRUnits.usiNumberOfUnits] OF UDINT;
	// Generated instance path of persistent variable
	Conveyors.Data: ARRAY [1..Conveyors.usiNumberOfUnits] OF Conveyor_Servo_Data;
	// Generated instance path of persistent variable
	Conveyors.DataBrink: ARRAY [1..Conveyors.usiNumberOfUnits] OF DataBrinkType;
	// Generated instance path of persistent variable
	Conveyors.DataReject: ARRAY [1..Conveyors.usiNumberOfUnits] OF Conveyor_Reject_Data;
	// Generated instance path of persistent variable
	Conveyors.coveredDistance: ARRAY [1..Conveyors.usiNumberOfUnits] OF UDINT;
	// Generated instance path of persistent variable
	Chains.Data: ARRAY [1..Chains.usiNumberOfUnits] OF ChainBase_Data;
	// Generated instance path of persistent variable
	Chains.DataProject: ARRAY [1..Chains.usiNumberOfUnits] OF Chain_WithCarrierPlates_Data;
	// Generated instance path of persistent variable
	Chains.DataBrink: ARRAY [1..Chains.usiNumberOfUnits] OF DataBrinkType;
	// Generated instance path of persistent variable
	Chains.coveredDistance: ARRAY [1..Chains.usiNumberOfUnits] OF UDINT;
	// Generated instance path of persistent variable
	Magazines.Data: ARRAY [1..Magazines.usiNumberOfUnits] OF Magazine_Data;
	// Generated instance path of persistent variable
	Magazines.DataMotors: ARRAY [1..Magazines.usiNumberOfUnits] OF MagazineMotors_Drawer_Data;
	// Generated instance path of persistent variable
	Magazines.DataBrink: ARRAY [1..Magazines.usiNumberOfUnits] OF MagazineMotors_Drawer_BrinkData;
	// Generated instance path of persistent variable
	Magazines.coveredDistance: ARRAY [1..Magazines.usiNumberOfUnits] OF ARRAY [PickPlaceAxesNames.A1..PickPlaceAxesNames.A2] OF UDINT;
	// Generated instance path of persistent variable
	InjectionMouldingMachine.Data: IMM_Data;
	// Generated instance path of persistent variable
	ProcessModules.XYControlData: ARRAY [1..ProcessModules.numberOfXYControls] OF XYControl_Data;
	// Generated instance path of persistent variable
	LabelSuppliers.Data: ARRAY [1..LabelSuppliers.usiNumberOfUnits] OF DrawerMagazine_Data;
	// Generated instance path of persistent variable
	VisionSystems.Data: ARRAY [1..VisionSystems.usiNumberOfUnits] OF VisionSystem_Base_Data;
	// Generated instance path of persistent variable
	VisionSystems.DataProject: ARRAY [1..VisionSystems.usiNumberOfUnits] OF VisionSystem_Mevisco_Data;
	// Generated instance path of persistent variable
	RejectStations.Data: ARRAY [1..RejectStations.usiNumberOfUnits] OF RejectStation_Base_Data;
	// Generated instance path of persistent variable
	RejectStations.DataProject: ARRAY [1..RejectStations.usiNumberOfUnits] OF RejectStation_WithBlowOff_Data;
	// Generated instance path of persistent variable
	BufferRacks.Data: ARRAY [1..BufferRacks.usiNumberOfUnits] OF BufferRack_Data;
	// Generated instance path of persistent variable
	BufferRacks.BufferStackStatus: ARRAY [1..BufferRacks.usiNumberOfUnits] OF StackStatusType;
	// Generated instance path of persistent variable
	BufferRacks.BufferStackIndex: USINT;
	// Generated instance path of persistent variable
	BoxInfeeds.Data: ARRAY [1..BoxInfeeds.usiNumberOfUnits] OF BoxInfeed_Default_DataType;
	// Generated instance path of persistent variable
	BoxCenterUnits.Data: ARRAY [1..BoxCenterUnits.usiNumberOfUnits] OF BoxCenterUnit_WithPneumatic_DataType;
	// Generated instance path of persistent variable
	BoxPushers.Data: ARRAY [1..BoxPushers.usiNumberOfUnits] OF BoxPusher_Default_DataType;
	// Generated instance path of persistent variable
	BoxOutfeeds.Data: ARRAY [1..BoxOutfeeds.usiNumberOfUnits] OF BoxOutfeed_Default_DataType;
END_VAR

%CLASS PERSISTENT
